TYPE EL2595_Data :
STRUCT
	{attribute addProperty Name "DOX Status"}
	DOXStatus : DOXStatusChannel;
	{attribute addProperty Name "DOX Control"}
	DOXControl : DOXControlCompactChannel;
END_STRUCT
END_TYPE

(* stored: Version 1.1.0.1, ProductVersion 3.1.4024.9
   DUT EL2595_Data: Id {4bdc2ffc-4690-03ce-36d5-d19eb2802069} *)
